RoboDK station: Bill_Dance_Demo.rdk

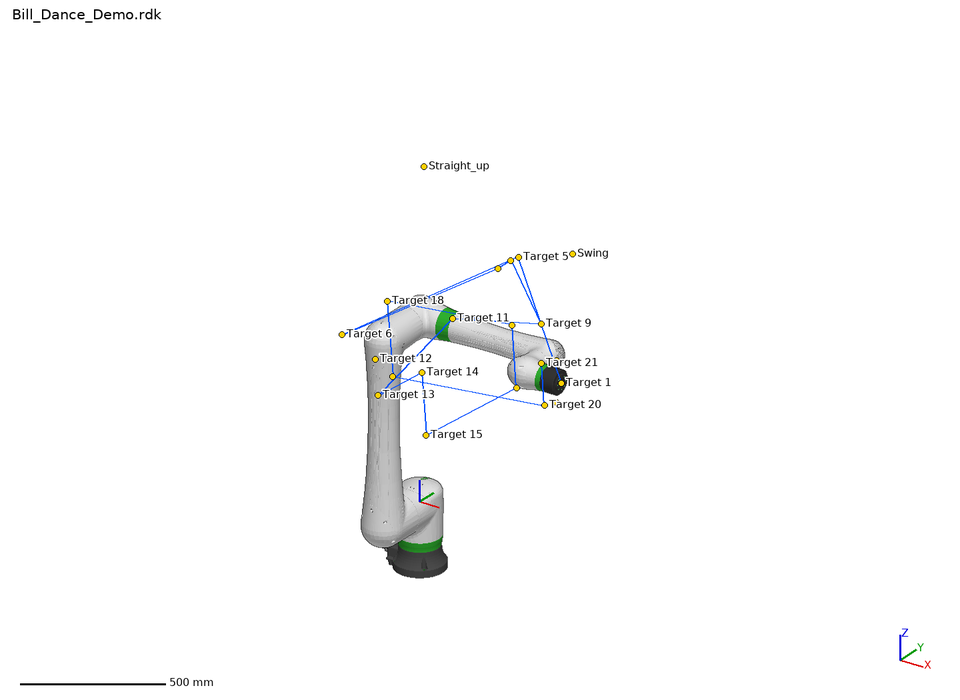
[picture v0: the station drawn from its stored meshes, robots at their saved joint values, targets as dots, program paths as lines]
Station Bill_Dance_Demo (saved by RoboDK 5.5.4). Poses are relative to the parent item; angles as X-Y-Z fixed-axis rotations.
Station parameters (name, value as stored): LIN64
  - frame Bill_Base at (0, 0, 245) mm
    - robot Fanuc CRX-10iA/L: 6 axes, payload 10 kg, reach 1418 mm, repeatability 0.05 mm, weight 40 kg
        modified DH rows (alpha deg, a mm, theta deg, d mm): 0, 0, 0, 245; -90, 0, -90, 0; 0, 710, 0, 0; -90, 0, 0, 540; 90, 0, 0, -150; -90, 0, 0, 160
        base shift (0, 0, -245) mm
        joint limits [-180, -180, -360, -190, -180, -190] to [180, 180, 430, 190, 180, 190]; home [0, 0, 0, 0, 0, 0]; saved at [0, 0, 0, 0, 0, 0]
    - target Target 1 (Cartesian target) at (700, -150, 710) mm, rotated rx 0 ry -48.49 rz -180 deg; joints [0, 4.066, -11.131, 0, 52.641, 0] of Fanuc CRX-10iA/L
    - target Target 2 (Cartesian target) at (700, -150, 710) mm, rotated rx -180 ry -54.48 rz 0 deg; joints [0, 3.069, 10.022, 0, -45.542, 0] of Fanuc CRX-10iA/L
    - target Target 3 (Cartesian target) at (700, -150, 710) mm, rotated rx -0.75 ry -66.26 rz -180 deg; joints [0.209, 1.357, -6.304, -1.886, 30.058, 1.717] of Fanuc CRX-10iA/L
    - target Target 4 (Cartesian target) at (700, -150, 710) mm, rotated rx 145.06 ry -44.05 rz 45.13 deg; joints [0, 3.165, 10.17, 0, -46.268, 30.62] of Fanuc CRX-10iA/L
    - target Target 5 (Cartesian target) at (518.38, -150, 1140.94) mm, rotated rx 0 ry -55.73 rz -180 deg; joints [0, -2.59, 39.239, 0, -4.974, 0] of Fanuc CRX-10iA/L
    - target Target 6 (Cartesian target) at (-221.33, -150, 636.99) mm, rotated rx 0 ry -55.73 rz -180 deg; joints [-150.216, -12.859, -29.903, 72.366, 154.484, -91.542] of Fanuc CRX-10iA/L
    - target Target 7 (Cartesian target) at (486.45, -227.04, 1119.19) mm, rotated rx 0 ry -55.73 rz -180 deg; joints [-21.2, -3.225, 48.288, -56.138, -21.095, 41.957] of Fanuc CRX-10iA/L
    - target Target 8 (Cartesian target) at (486.45, -150, 1119.19) mm, rotated rx -4.3 ry 55.62 rz -5.21 deg; joints [0, -6.324, 36.794, 0, -2.528, 182.937] of Fanuc CRX-10iA/L
    - target Target 9 (Cartesian target) at (623.02, -162.44, 918.73) mm, rotated rx -4.3 ry 55.62 rz -5.21 deg; joints [-1.451, 64.254, 105.902, -1.263, -71.632, -177.482] of Fanuc CRX-10iA/L
    - target Target 10 (Cartesian target) at (623.02, -162.44, 918.73) mm, rotated rx -159.3 ry 83.12 rz -161.09 deg; joints [-0.877, 54.843, 101.883, 1.1, -108.315, -177.33] of Fanuc CRX-10iA/L
    - target Target 11 (Cartesian target) at (245.54, -155.29, 830.18) mm, rotated rx -19.92 ry 82.86 rz -21.44 deg; joints [-0.998, -34.413, 24.374, 1.215, -17.67, -178.671] of Fanuc CRX-10iA/L
    - target Target 12 (Cartesian target) at (232.75, -598.06, 848.95) mm, rotated rx -19.92 ry 82.86 rz -21.44 deg; joints [-83.478, 4.19, 28.103, -92.259, -79.904, -114.997] of Fanuc CRX-10iA/L
    - target Target 13 (Cartesian target) at (248.07, -604.08, 717.49) mm, rotated rx -19.92 ry 82.86 rz -21.44 deg; joints [-82.63, 3.757, 14.492, -94.388, -79.903, -101.148] of Fanuc CRX-10iA/L
    - target Target 14 (Cartesian target) at (255.31, -353.57, 706.87) mm, rotated rx -19.92 ry 82.86 rz -21.44 deg; joints [-75.492, -16.159, 16.151, -92.195, -72.934, -102.441] of Fanuc CRX-10iA/L
    - target Target 15 (Cartesian target) at (281.85, -363.99, 479.16) mm, rotated rx -19.92 ry 82.86 rz -21.44 deg; joints [-74.961, -10.301, -9.854, -99.714, -75.142, -75.465] of Fanuc CRX-10iA/L
    - target Target 16 (Cartesian target) at (296.86, 155.94, 457.12) mm, rotated rx -19.92 ry 82.86 rz -21.44 deg; joints [57.041, -26.277, -5.492, -78.894, 59.556, -97.979] of Fanuc CRX-10iA/L
    - target Target 17 (Cartesian target) at (270.35, 166.35, 684.61) mm, rotated rx -19.92 ry 82.86 rz -21.44 deg; joints [51.284, -30.026, 20.645, -97.441, 52.773, -66.672] of Fanuc CRX-10iA/L
    - target Target 18 (Cartesian target) at (-262.53, 179.08, 621.92) mm, rotated rx -19.92 ry 82.86 rz -21.44 deg; joints [168.56, -7.584, 1.585, -50.375, 166.969, -48.384] of Fanuc CRX-10iA/L
    - target Target 19 (Cartesian target) at (-230.68, 166.57, 348.65) mm, rotated rx -19.92 ry 82.86 rz -21.44 deg; joints [146.094, 1.078, -29.696, -120.395, 141.737, -128.581] of Fanuc CRX-10iA/L
    - target Target 20 (Cartesian target) at (417.67, 151.08, 424.93) mm, rotated rx -19.92 ry 82.86 rz -21.44 deg; joints [42.569, -15.273, -15.776, -65.998, 48.969, -115.283] of Fanuc CRX-10iA/L
    - target Target 21 (Cartesian target) at (399.84, 158.08, 577.84) mm, rotated rx -19.92 ry 82.86 rz -21.44 deg; joints [36.162, -21.572, 5.084, -85.6, 37.359, -87.959] of Fanuc CRX-10iA/L
    - target Home (Cartesian target) at (700, -150, 710) mm, rotated rx 0 ry -90 rz -180 deg; joints [0, 0, 0, 0, 0, 0] of Fanuc CRX-10iA/L
    - target Wave_Down (Cartesian target) at (678.56, -150, 630) mm, rotated rx -180 ry -60 rz 0 deg; joints [0, 0, 0, 0, -30, 0] of Fanuc CRX-10iA/L
    - target Wave_up (Cartesian target) at (678.56, -150, 790) mm, rotated rx 0 ry -60 rz -180 deg; joints [0, 0, 0, 0, 30, 0] of Fanuc CRX-10iA/L
    - target Swing (Cartesian target) at (150, 700, 710) mm, rotated rx 0 ry -90 rz -90 deg; joints [90, 0, 0, 0, 0, 0] of Fanuc CRX-10iA/L
    - target Straight_up (Cartesian target) at (122.31, -150, 1375.32) mm, rotated rx 0 ry -21.62 rz -180 deg; joints [0, -6.37, 74.74, 0, -6.36, 0] of Fanuc CRX-10iA/L
  - Python program Dance_Bill (listed below)
  - Python program Prog2 (listed below)
  - program Prog3 (21 instructions, listed below)
  - Python program crx10_sync (listed below)
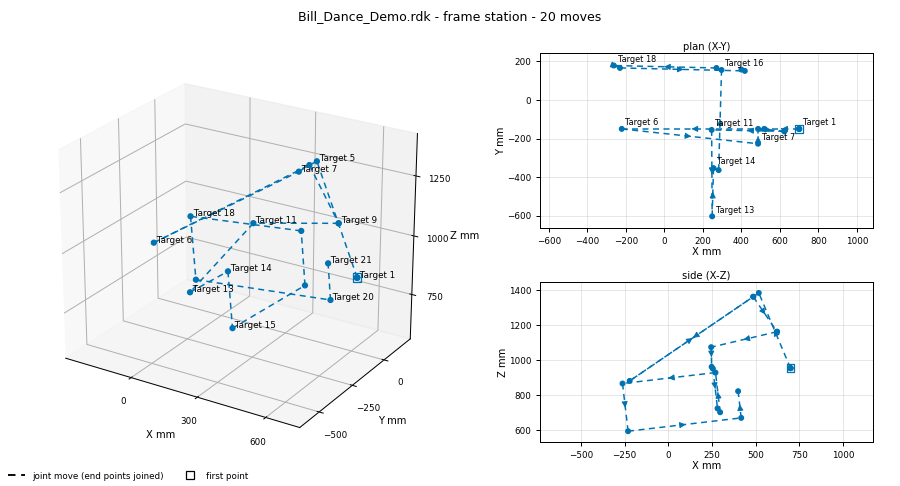
[picture p0: tool path of Bill_Dance_Demo.rdk in frame station, 20 of 20 moves have a stored position in this frame; points joined in program order, loops and branches not executed]

--- Python program Dance_Bill ---
import time
import random as rand

from robodk.robolink import *                  # import the robolink library
RDK = Robolink()                        # connect to the RoboDK API (RoboDK starts if it has not started

robots = RDK.ItemList(ITEM_TYPE_ROBOT)
print(robots)


# tool  = RDK.Item('SCHUNK- 1321170 Co-act EGP-C 40-N-N-KTOE_ 0')                # Get an item named Tool (name in the RoboDK station tree)

robot = RDK.Item('', ITEM_TYPE_ROBOT)   # Get the first available robot


robot.Connect()
RDK.setRunMode(RUNMODE_RUN_ROBOT)
#RDK.setRunMode(RUNMODE_SIMULATE)
#frame = RDK.ItemUserPick('Select a reference frame', ITEM_TYPE_FRAME)   # Promt the user to select a reference frame
frame = RDK.Item('Frame 2', ITEM_TYPE_FRAME)

robot.setPoseFrame(frame)
# robot.setPoseTool(tool)
rand_speed = rand.randrange(20, 100, 5)

# robot.setSpeed(1500)


def dance():
	robot.setSpeed(1500, speed_joints = rand_speed)
	target = RDK.Item('Target 1', ITEM_TYPE_TARGET)
	robot.MoveJ(target)

	target = RDK.Item('Target 2', ITEM_TYPE_TARGET)   # Get a target called "turn1"
	robot.MoveJ(target)             # Move the robot to the target using the selected reference frame


	robot.setSpeed(1500, speed_joints = rand_speed)
	target = RDK.Item('Target 3', ITEM_TYPE_TARGET)   # Get a target called "home"
	robot.MoveJ(target)

	#robot.setSpeed(1500, speed_joints = 20)
	target = RDK.Item('Target 4', ITEM_TYPE_TARGET)
	robot.MoveJ(target)

	target = RDK.Item('Target 5', ITEM_TYPE_TARGET)   # Get a target called "turn1"
	robot.MoveJ(target)             # Move the robot to the target using the selected reference frame


	robot.setSpeed(1500, speed_joints = rand_speed)
	target = RDK.Item('Target 6', ITEM_TYPE_TARGET)   # Get a target called "home"
	robot.MoveJ(target)

	robot.setSpeed(1500, speed_joints = rand_speed)
	target = RDK.Item('Target 7', ITEM_TYPE_TARGET)
	robot.MoveJ(target)

	target = RDK.Item('Target 8', ITEM_TYPE_TARGET)   # Get a target called "turn1"
	robot.MoveJ(target)             # Move the robot to the target using the selected reference frame


	robot.setSpeed(1500, speed_joints = rand_speed)
	target = RDK.Item('Target 9', ITEM_TYPE_TARGET)   # Get a target called "home"
	robot.MoveJ(target)

	target = RDK.Item('Target 10', ITEM_TYPE_TARGET)   # Get a target called "turn1"
	robot.MoveJ(target)             # Move the robot to the target using the selected reference frame


	robot.setSpeed(1500, speed_joints = rand_speed)
	target = RDK.Item('Target 11', ITEM_TYPE_TARGET)   # Get a target called "home"
	robot.MoveJ(target)

	robot.setSpeed(1500, speed_joints = rand_speed)
	target = RDK.Item('Target 12', ITEM_TYPE_TARGET)
	robot.MoveJ(target)

	target = RDK.Item('Target 13', ITEM_TYPE_TARGET)   # Get a target called "turn1"
	robot.MoveJ(target)             # Move the robot to the target using the selected reference frame


	robot.setSpeed(1500, speed_joints = rand_speed)
	target = RDK.Item('Target 14', ITEM_TYPE_TARGET)   # Get a target called "home"
	robot.MoveJ(target)

	robot.setSpeed(1500, speed_joints = rand_speed)
	target = RDK.Item('Target 15', ITEM_TYPE_TARGET)   # Get a target called "home"
	robot.MoveJ(target)

	robot.setSpeed(1500, speed_joints = rand_speed)
	target = RDK.Item('Target 16', ITEM_TYPE_TARGET)
	robot.MoveJ(target)

	target = RDK.Item('Target 17', ITEM_TYPE_TARGET)   # Get a target called "turn1"
	robot.MoveJ(target)             # Move the robot to the target using the selected reference frame


	robot.setSpeed(1500, speed_joints = rand_speed)
	target = RDK.Item('Target 18', ITEM_TYPE_TARGET)   # Get a target called "home"
	robot.MoveJ(target)

	robot.setSpeed(1500, speed_joints = rand_speed)
	target = RDK.Item('Target 19', ITEM_TYPE_TARGET)   # Get a target called "home"
	robot.MoveJ(target)

	robot.setSpeed(1500, speed_joints = rand_speed)
	target = RDK.Item('Target 20', ITEM_TYPE_TARGET)
	robot.MoveJ(target)

	robot.setSpeed(1500, speed_joints = 50)
	target = RDK.Item('Target 21', ITEM_TYPE_TARGET)   # Get a target called "turn1"
	robot.MoveJ(target)             # Move the robot to the target using the selected reference frame
for i in range(0,1):
	print("Run: ", i)
	dance()

--- Python program Prog2 ---
# Type help("robodk.robolink") or help("robodk.robomath") for more information
# Press F5 to run the script
# Documentation: https://robodk.com/doc/en/RoboDK-API.html
# Reference:     https://robodk.com/doc/en/PythonAPI/robodk.html
# Note: It is not required to keep a copy of this file, your Python script is saved with your RDK project

# You can also use the new version of the API:
from robodk import robolink    # RoboDK API
from robodk import robomath    # Robot toolbox
RDK = robolink.Robolink()

# Forward and backwards compatible use of the RoboDK API:
# Remove these 2 lines to follow python programming guidelines
from robodk import *      # RoboDK API
from robolink import *    # Robot toolbox
# Link to RoboDK
# RDK = Robolink()

# Notify user:
print('To edit this program:\nright click on the Python program, then, select "Edit Python script"')

# Program example:
item = RDK.Item('base')
if item.Valid():
    print('Item selected: ' + item.Name())
    print('Item posistion: ' + repr(item.Pose()))

print('Items in the station:')
itemlist = RDK.ItemList()
print(itemlist)

# Provoking an exception will display the console output if you run this script from RoboDK
raise Exception('Program not edited.')

--- program Prog3 (robot Fanuc CRX-10iA/L) ---
  Set Ref.: Bill_Base
  MoveJ (Target 1)
  MoveJ (Target 2)
  MoveJ (Target 3)
  MoveJ (Target 4)
  MoveJ (Target 5)
  MoveJ (Target 6)
  MoveJ (Target 7)
  MoveJ (Target 8)
  MoveJ (Target 9)
  MoveJ (Target 10)
  MoveJ (Target 11)
  MoveJ (Target 13)
  MoveJ (Target 14)
  MoveJ (Target 15)
  MoveJ (Target 16)
  MoveJ (Target 17)
  MoveJ (Target 18)
  MoveJ (Target 19)
  MoveJ (Target 20)
  MoveJ (Target 21)

--- Python program crx10_sync ---
# imports
import random as rand
from threading import RLock
from robodk.robolink import *           # import the robolink library
# connect to the RoboDK API (RoboDK starts if it has not started)
RDK = Robolink()

# common variables - config
mqtt_err = False
robot_name = "bill"
start_sync = False
lock = RLock()

try:
    import paho.mqtt.client as paho
    from paho import mqtt
except Exception as e:
    print("Error: please install 'paho.mqtt.client' module.")
    mqtt_err = True

# ---------------------------
#
# mqtt callbacks
#
# ---------------------------


def on_connect(client, userdata, flags, rc, properties=None):
    if rc == 0:
        print(f'connected successfuly code={rc}')


def on_subscribe(client, userdata, mid, granted_qos, properties=None):
    print(f'Subscribed: {mid} {granted_qos}')


def on_publish(client, userdata, mid, properties=None):
    print(f'mid: {mid}')


def on_message(client, userdata, msg):
    print("message received")
    message_string = msg.payload.decode("ascii")

    print(f'\ntopic: {msg.topic}')
    print(f'{message_string}')

    if msg.topic == "synchronize" and robot_name not in message_string:
        print('received message from other robot')
        with lock:
            global start_sync
            start_sync = True
    else:
        print('received message from self')


def on_disconnect(client, userdata, rc, properties=None):
    if rc == paho.MQTT_ERR_SUCCESS:
        print("Disconnected successfully")
    else:
        print("Unexpected disconnect")

# ---------- connecting to mqtt broker


def connect_local_MQTT():
    print("start connecting")
    client_id = robot_name
    localMQTT = paho.Client(client_id)

    # set up call backs
    localMQTT.on_connect = on_connect
    ip_addr = "453e51c107604519a5fd673fd39f1313.s1.eu.hivemq.cloud"
    port = 8883
    username = "student"
    password = "cs383_students"
    # connect
    localMQTT.tls_set(tls_version=mqtt.client.ssl.PROTOCOL_TLS)
    localMQTT.username_pw_set(username, password)
    localMQTT.connect(host=ip_addr, port=port)

    # more callbacks
    localMQTT.on_message = on_message
    localMQTT.on_subscribe = on_subscribe
    localMQTT.on_disconnect = on_disconnect
    localMQTT.on_publish = on_publish

    return localMQTT


def publishMessage(topic, message):
    print("starting to publish")

    clientname = client._client_id
    clientname = clientname.decode(("ascii"))
    new_msg = f"{clientname}: {message}"
    client.publish(topic, new_msg, qos=1)

# -----------------
#
# robodk code
#
# -----------------


def dance(rand_speed):
    robot.setSpeed(1500, speed_joints=rand_speed)
    target = RDK.Item('Target 1', ITEM_TYPE_TARGET)
    robot.MoveJ(target)

    # Get a target called "turn1"
    target = RDK.Item('Target 2', ITEM_TYPE_TARGET)
    # Move the robot to the target using the selected reference frame
    robot.MoveJ(target)

    robot.setSpeed(1500, speed_joints=rand_speed)
    # Get a target called "home"
    target = RDK.Item('Target 3', ITEM_TYPE_TARGET)
    robot.MoveJ(target)

    # robot.setSpeed(1500, speed_joints = 20)
    target = RDK.Item('Target 4', ITEM_TYPE_TARGET)
    robot.MoveJ(target)

    # Get a target called "turn1"
    target = RDK.Item('Target 5', ITEM_TYPE_TARGET)
    # Move the robot to the target using the selected reference frame
    robot.MoveJ(target)

    robot.setSpeed(1500, speed_joints=rand_speed)
    # Get a target called "home"
    target = RDK.Item('Target 6', ITEM_TYPE_TARGET)
    robot.MoveJ(target)

    robot.setSpeed(1500, speed_joints=rand_speed)
    target = RDK.Item('Target 7', ITEM_TYPE_TARGET)
    robot.MoveJ(target)

    # Get a target called "turn1"
    target = RDK.Item('Target 8', ITEM_TYPE_TARGET)
    # Move the robot to the target using the selected reference frame
    robot.MoveJ(target)

    robot.setSpeed(1500, speed_joints=rand_speed)
    # Get a target called "home"
    target = RDK.Item('Target 9', ITEM_TYPE_TARGET)
    robot.MoveJ(target)

    # Get a target called "turn1"
    target = RDK.Item('Target 10', ITEM_TYPE_TARGET)
    # Move the robot to the target using the selected reference frame
    robot.MoveJ(target)

    robot.setSpeed(1500, speed_joints=rand_speed)
    # Get a target called "home"
    target = RDK.Item('Target 11', ITEM_TYPE_TARGET)
    robot.MoveJ(target)

    robot.setSpeed(1500, speed_joints=rand_speed)
    target = RDK.Item('Target 12', ITEM_TYPE_TARGET)
    robot.MoveJ(target)

    # Get a target called "turn1"
    target = RDK.Item('Target 13', ITEM_TYPE_TARGET)
    # Move the robot to the target using the selected reference frame
    robot.MoveJ(target)

    robot.setSpeed(1500, speed_joints=rand_speed)
    # Get a target called "home"
    target = RDK.Item('Target 14', ITEM_TYPE_TARGET)
    robot.MoveJ(target)

    robot.setSpeed(1500, speed_joints=rand_speed)
    # Get a target called "home"
    target = RDK.Item('Target 15', ITEM_TYPE_TARGET)
    robot.MoveJ(target)

    robot.setSpeed(1500, speed_joints=rand_speed)
    target = RDK.Item('Target 16', ITEM_TYPE_TARGET)
    robot.MoveJ(target)

    # Get a target called "turn1"
    target = RDK.Item('Target 17', ITEM_TYPE_TARGET)
    # Move the robot to the target using the selected reference frame
    robot.MoveJ(target)

    robot.setSpeed(1500, speed_joints=rand_speed)
    # Get a target called "home"
    target = RDK.Item('Target 18', ITEM_TYPE_TARGET)
    robot.MoveJ(target)

    robot.setSpeed(1500, speed_joints=rand_speed)
    # Get a target called "home"
    target = RDK.Item('Target 19', ITEM_TYPE_TARGET)
    robot.MoveJ(target)

    robot.setSpeed(1500, speed_joints=rand_speed)
    target = RDK.Item('Target 20', ITEM_TYPE_TARGET)
    robot.MoveJ(target)

    robot.setSpeed(1500, speed_joints=rand_speed)
    # Get a target called "turn1"
    target = RDK.Item('Target 21', ITEM_TYPE_TARGET)
    robot.MoveJ(target)

    robot.setSpeed(1500, speed_joints=100)
    # Get a target called "turn1"
    target = RDK.Item('Home', ITEM_TYPE_TARGET)
    robot.MoveJ(target)


def start_robodk(robolink, runmode, frame_name):
    robot = robolink.Item('', ITEM_TYPE_ROBOT)
    robot.Connect()
    robolink.setRunMode(runmode)

    frame = robolink.Item(frame_name, ITEM_TYPE_FRAME)
    robot.setPoseFrame(frame)

    return robot


def move_robot(robot, tgt_names, lin_speed=1500, j_speed=180, loop=1):

    for i in range(0, len(tgt_names)*loop):             # move through targets
        robot.setSpeed(speed_linear=lin_speed,
                       speed_joints=j_speed)                  # set speed
        target = RDK.Item(tgt_names[i % len(tgt_names)], ITEM_TYPE_TARGET)
        robot.MoveJ(target)

# ---------main program----------


robot = start_robodk(RDK, RUNMODE_RUN_ROBOT, 'Bill_Base')

if not mqtt_err:
    client = connect_local_MQTT()
    client.subscribe("#")

    client.loop_start()

    print(f'started listening program for {robot_name}')

    # put robot code here
    rand_speed = rand.randrange(20, 100, 5)
    # move_robot(robot, ['squat_down'], j_speed=50)
    dance(rand_speed)

    publishMessage('synchronize', 'ready')

    while not start_sync:
        # wait for other robot to be done
        pass

    print(f'now starting synchronized swimming program')

    # synchronized robot code here
    move_robot(robot, ['Home'])
    move_robot(robot, ['Wave_Down', 'Wave_up'], loop=2)
    move_robot(robot, ['Swing', 'Straight_up'])
    move_robot(robot, ['Home'])

    client.loop_stop()
    client.disconnect()
